Omron Sysmac Studio project OEEF_FS_lib_1_3_7 (Sysmac Studio 1.60.0.64010, LibraryProject)

# Controller new_Controller_0: NX1P2-1040DT1 version 1.21
Task PrimaryTask (priority 4, period or condition 2000): Programme0

TYPE nsAxisControl\eMoveMode : (Relative := 0, Absolute := 1); END_TYPE
TYPE nsAxisControl\eCurveType : (Poly5 := 0, Poly3 := 1, Straight := 2, NoCurve := 9999); END_TYPE
TYPE nsAxisControl\eTypeOfCmd : (CancelMC_Sync := -5, CancelCam := -3, CancelTrack := -2, NoCde := 9999, PolyMvt := 1, Track := 2, Cam := 3, WarmStart := 4, MC_Sync := 5); END_TYPE
TYPE nsAxisControl\stAxisControl : STRUCT
    MasterPosition : nsAxisControl\stMasterPosition;
    MasterAxis : _sAXIS_REF;
    Move : nsAxisControl\stMove;
    Track : nsAxisControl\stTrack;
    Cam : nsAxisControl\stCam;
    Flags : nsAxisControl\stFlags;
    Monitoring : nsAxisControl\stMonitoring;
    MC_MoveJog : nsAxisControl\stMC_MoveJog;
    MC_SetPosition : nsAxisControl\stMC_SetPosition;
    MC_Power : nsAxisControl\stMC_Power;
    MC_Home : nsAxisControl\stMC_Home;
END_STRUCT END_TYPE
TYPE nsAxisControl\stMC_Power : STRUCT
    Enable : BOOL;
    Status : BOOL;
    Busy : BOOL;
    Error : BOOL;
    ErrorID : WORD;
END_STRUCT END_TYPE
TYPE nsAxisControl\stMC_MoveJog : STRUCT
    PositiveEnable : BOOL;
    NegativeEnable : BOOL;
    Velocity : LREAL;
    Acceleration : LREAL;
    Deceleration : LREAL;
    Busy : BOOL;
    CommandAborted : BOOL;
    Error : BOOL;
    ErrorID : WORD;
END_STRUCT END_TYPE
TYPE nsAxisControl\stMC_SetPosition : STRUCT
    Execute : BOOL;
    Position : LREAL;
    ReferenceType : _eMC_REFERENCE_TYPE;
    Relative : BOOL;
    ExecutionMode : _eMC_EXECUTION_MODE;
    Done : BOOL;
    Busy : BOOL;
    CommandAborted : BOOL;
    Error : BOOL;
    ErrorID : WORD;
END_STRUCT END_TYPE
TYPE nsAxisControl\stMC_Home : STRUCT
    Execute : BOOL;
    Done : BOOL;
    Busy : BOOL;
    CommandAborted : BOOL;
    Error : BOOL;
    ErrorID : WORD;
END_STRUCT END_TYPE
TYPE nsAxisControl\stMasterPosition : STRUCT
    NotFrom_sAXIS_REF : BOOL;
    ExternalVariable : LREAL;
END_STRUCT END_TYPE
TYPE nsAxisControl\stMove : STRUCT
    Pos : LREAL;
    Dist : LREAL;
    Tim : LREAL;
    Accel : LREAL;
    Decel : LREAL;
    PolyType : nsAxisControl\eCurveType;
    Mode : nsAxisControl\eMoveMode;
    SetT_In : LREAL;
    SetT_Out : LREAL;
    T_InDone : BOOL;
    T_OutDone : BOOL;
    Exe : BOOL;
END_STRUCT END_TYPE
TYPE nsAxisControl\stTrack : STRUCT
    TrackPos : LREAL;
    Tim : LREAL;
    TimStop : LREAL;
    SetT_In : LREAL;
    T_InDone : BOOL;
    Exe : BOOL;
    Cancel : BOOL;
END_STRUCT END_TYPE
TYPE nsAxisControl\stCam : STRUCT
    Profile : ARRAY[0..10] OF nsAxisControl\stNodes;
    MasterOffset : LREAL;
    SlaveOffset : LREAL;
    ProfileToApply : INT;
    WarmStartSlavePos : LREAL;
    WarmStartSlavePosRequest : BOOL;
    Exe : BOOL;
    Cancel : BOOL;
END_STRUCT END_TYPE
TYPE nsAxisControl\stNodes : STRUCT
    Node : ARRAY[0..10] OF nsAxisControl\stNode;
END_STRUCT END_TYPE
TYPE nsAxisControl\stNode : STRUCT
    MasterAxisPos : LREAL;
    SlaveAxisPos : LREAL;
    CurveTypeBefore : nsAxisControl\eCurveType;
    StartingSlope : LREAL;
    EndingSlope : LREAL;
END_STRUCT END_TYPE
TYPE nsAxisControl\stFlags : STRUCT
    Done : BOOL;
    Synchronised : BOOL;
END_STRUCT END_TYPE
TYPE nsAxisControl\stMonitoring : STRUCT
    PositioningCmd : LREAL;
    CurrentProfile : INT;
    CurrentSegment : INT;
    TypeOfCmd : nsAxisControl\eTypeOfCmd;
END_STRUCT END_TYPE
TYPE nsAxisControl\eReferenceType : (mcCommand := 0, mcFeedback := 1); END_TYPE

PROGRAM Programme0

(* Section Section0: ladder, written here as Structured Text *)
END_PROGRAM

FUNCTION fPolyTimesNeeded : BOOL
(* - Time needed to achieve a movement depending of the curve type and the acceleration or the speed fixed. To do for instance a speed or an acceleration limit. *)
VAR_INPUT
    CurveType : nsAxisControl\eCurveType;
    Distance : LREAL;
    AccDefined : LREAL;
    SpeedDefined : LREAL;
END_VAR
VAR_OUTPUT
    TNeededToAcc : LREAL;
    TNeededToSpeed : LREAL;
END_VAR
(*
*******************************************
*		  Calcule le temps nécessaire			*
*	 pour effectuer un trajet avec une		*
*	accélération ou une vitesse définie		*
*******************************************
*)

CASE CurveType OF
	
	Poly5 :
	// AccDefined exprimée en unité/sec2
	TNeededToAcc:=SQRT(5.8*Distance/AccDefined);

	// SpeedDefined exprimée en unité/sec
	TNeededToSpeed:=1.9*Distance/SpeedDefined;
	
	Poly3 :
	// AccDefined exprimée en unité/sec2
	TNeededToAcc:=SQRT(6*Distance/AccDefined);

	// SpeedDefined exprimée en unité/sec
	TNeededToSpeed:=1.5*Distance/SpeedDefined;
	
END_CASE;
END_FUNCTION

FUNCTION fTicksQCalc : LINT
(* - Calculation of the quantity of ticks depending of the time of the movement *)
VAR
    TaskPeriod_msec : LINT;
END_VAR
VAR_INPUT
    TimeMvt : LREAL;
END_VAR
(*
*******************************************
*		  			Calcule le nombre				*
*	 					de cycles cpu					*
*******************************************
*)

// Suivant le temps de cycle de la tâche principale
TaskPeriod_msec:= TimeToNanoSec(GetMyTaskInterval())/1000000;

// Suivant le temps du mouvement en secondes
fTicksQCalc:=LREAL_TO_LINT(TimeMvt*1000)/TaskPeriod_msec;
END_FUNCTION

FUNCTION fPoly5 : LREAL
(* - Polynomial of the 5th order *)
VAR
    a : LREAL;
    b : LREAL;
    c : LREAL;
    d : LREAL;
    e : LREAL;
    f : LREAL;
    K : LREAL;
    xSq : LREAL;
END_VAR
VAR_INPUT
    v0 : LREAL;  (* Vitesse initiale *)
    v1 : LREAL;  (* Vitesse finale *)
    a0 : LREAL;
    a1 : LREAL;
    x : LREAL;
    Offset : LREAL;
    TargetDist : LREAL;
END_VAR
(*
*******************************************
*		  				Polynôme 5						*
*******************************************
*)

// Coéficients 
a:=6.0-3.0*(v0+v1)+((a1-a0)/2.0);
b:=-15.0+8.0*v0+7.0*v1+(3.0*a0/2.0)-a1;
c:=10.0-6.0*v0-4.0*v1-(3.0*a0/2.0)+(a1/2.0);
d:=a0/2.0;
e:=v0;
f:=Offset;
K:=TargetDist;

// Position=ax5+bx4+cx3+dx2+ex+f
fPoly5:=f+(K*(a*(x**5)+b*(x**4)+c*(x**3)+d*(x**2)+e*x));
END_FUNCTION

FUNCTION fPoly3 : LREAL
(* - Polynomial of the 3th order *)
VAR
    a : LREAL;
    b : LREAL;
    c : LREAL;
    d : LREAL;
    K : LREAL;
    xSq : LREAL;
END_VAR
VAR_INPUT
    v0 : LREAL;  (* Vitesse initiale *)
    v1 : LREAL;  (* Vitesse finale *)
    x : LREAL;
    Offset : LREAL;
    TargetDist : LREAL;
END_VAR
(*
*******************************************
*		  				Polynôme 3						*
*******************************************
*)

// Coéficients 
a:=-2.0+v0+v1;
b:=3.0-2.0*v0-v1;
c:=v0;
d:=Offset;
K:=TargetDist;

// Position=ax3+bx2+cx+d
fPoly3:=d+(K*(a*(x**3)+b*(x**2)+c*x));
END_FUNCTION

FUNCTION fStraight : LREAL
(* - Straight *)
VAR
    a : LREAL;
    b : LREAL;
END_VAR
VAR_INPUT
    x : LREAL;
    Offset : LREAL;
    TargetDist : LREAL;
END_VAR
(*
*******************************************
*		  					Droite							*
*******************************************
*)

// Coéficients 
a:=TargetDist;
b:=Offset;

// Position=ax+b
fStraight:=a*x+b;
END_FUNCTION

FUNCTION fAtan2 : LREAL
(* - Arc tangent on four quadrants *)
VAR
    PI : LREAL := 3.14159265358979;
END_VAR
VAR_INPUT
    x : LREAL;
    y : LREAL;
END_VAR
(*
*******************************************
*  Calcule l'arc tangente (angle en rad)	*
*  d'un point [x,y] dans les 4 quadrants	*
*******************************************
*)

IF x>0 THEN
	fAtan2:=ATAN(y/x);
ELSIF x<0 AND y>=0 THEN
	fAtan2:=ATAN(y/x)+PI;
ELSIF x<0 AND y<0 THEN
	fAtan2:=ATAN(y/x)-PI;
ELSIF x=0 AND y>0 THEN
	fAtan2:=PI/2;
ELSIF x=0 AND y<0 THEN
	fAtan2:=-PI/2;
ELSIF x=0 AND y=0 THEN
	fAtan2:=0.0; // Non défini
END_IF;
END_FUNCTION

FUNCTION_BLOCK AxisControl
(* - Cam on fly (multi-profiles) / - Warm start / - Polynomial moves / - Conveyor tracking / - Blending (T_In & T_Out) *)
VAR
    FBi_SyncMov : MC_SyncMoveAbsolute;
    FBi_SyncStop : MC_Stop;
    FBe_SetPosition : MC_SetPosition;
    FBe_Home : MC_Home;
    FBi_SyncMovVel : MC_SyncMoveVelocity;
    FBi_ReadAxisMasterParam : MC_ReadAxisParameter;
    FBi_ReadAxisSlaveParam : MC_ReadAxisParameter;
    FBe_Power : MC_Power;
    Edge1 : R_TRIG;
    Edge2 : R_TRIG;
    Edge3 : R_TRIG;
    Edge4 : R_TRIG;
    Edge5 : R_TRIG;
    Edge6 : R_TRIG;
    Edge10 : R_TRIG;
    TypeOfCmd : nsAxisControl\eTypeOfCmd;
    TargetDist : LREAL;
    UpExecMvt : BOOL;
    UpExecTrack : BOOL;
    UpExecCam : BOOL;
    UpCancelTrack : BOOL;
    Phase : INT;
    Tick : LINT;
    TicksQ : LINT;
    Offset : LREAL;
    x : LREAL;
    v0 : LREAL;  (* Vitesse initiale *)
    v1 : LREAL;  (* Vitesse finale *)
    DistStop : LREAL;
    UpCancelCam : BOOL;
    MasterDistDone : LREAL;
    a1 : LREAL;
    a0 : LREAL;
    FBe_MovJog : MC_MoveJog;
    MemPosAxis : LREAL;
    ReadAxisMasterPParam : _sAXIS_PARAM;
    ReadAxisSlavePParam : _sAXIS_PARAM;
    CamSettingError : BOOL;
    NodesNbMax : INT;
    Loop : INT;
    X0 : LREAL;
    X1 : LREAL;
    Y0 : LREAL;
    Y1 : LREAL;
    SegmentPolyType : nsAxisControl\eCurveType;
    MasterDist : LREAL;
    SegmentsNb : INT;
    NodesNb : INT;
    UpWarmStartPosReq : BOOL;
    WarmStartCalculation : BOOL;
    v1CamSetting : LREAL;
    v0CamSetting : LREAL;
    a0CamSetting : LREAL;
    a1CamSetting : LREAL;
    ScannedSeg : INT;
    SetPositionErr : BOOL;
    SetPositionErrID : WORD;
    CurrentProfile : INT := 0;
    ProfilesNb : INT;
    ProfilesNbMax : INT;
    UpCamBeginning : BOOL;
    CamSettingErrorType : STRING[50];
    Gen : LREAL;
    Conveyor_Pos : LREAL;
    TaskPeriod_msec_LREAL : LREAL;
    MasterPosition : LREAL;
    TickSetT_In : LINT;
    TickSetT_Out : LINT;
    memSegmentNb : INT;
    memPosition : LREAL;
    SlaveMinPos : LREAL;
    SlaveMaxPos : LREAL;
    SlaveCountMode : _eMC_COUNT_MODE;
    MasterModulo : LREAL;
    ReadAxisDelay : TON;
    SlaveModulo : LREAL;
    CurrentSegment : INT;
    CmdPos : LREAL;
    TargetSpeed : LREAL;
    FBi_dx : FB_dx_Codeur_V2;
    MasterMinPos : LREAL;
    MasterMaxPos : LREAL;
    dx : LREAL;
    MemSpeedAxis : LREAL;
    MemActPos : LREAL;
    TrackStopDelay : TON;
END_VAR
VAR_INPUT
    Reset : BOOL;
    ExternalError : BOOL;
END_VAR
VAR_OUTPUT
    Error : BOOL;
END_VAR
VAR_IN_OUT CONSTANT
    Axis : _sAXIS_REF;
END_VAR
VAR_IN_OUT
    IO : nsAxisControl\stAxisControl;
END_VAR
VAR_OUTPUT
    ErrorMsg : STRING[80];
END_VAR
(*
*******************************************
*					OEEF - F.SIMON					*
*******************************************
*)


(*
*******************************************
*	 		Bits fronts de statuts : RAZ			*
*******************************************
*)
IF IO.Flags.Done THEN
	IO.Flags.Done:=FALSE;
END_IF;

IF IO.Move.T_InDone THEN
	IO.Move.T_InDone:=FALSE;
END_IF;

IF IO.Move.T_OutDone THEN
	IO.Move.T_OutDone:=FALSE;
END_IF;

IF IO.Track.T_InDone THEN
	IO.Track.T_InDone:=FALSE;
END_IF;


(*
*******************************************
*						Axe maître						*
*******************************************
*)
// Type
IF IO.MasterPosition.NotFrom_sAXIS_REF THEN
	MasterPosition:=IO.MasterPosition.ExternalVariable;
ELSE
	MasterPosition:=IO.MasterAxis.Act.Pos;
END_IF;

// Offset
MasterModulo:=(ReadAxisSlavePParam.PosCount.ModuloMaxPosVal-ReadAxisSlavePParam.PosCount.ModuloMinPosVal);
IF IO.Cam.MasterOffset<0 THEN
	MasterPosition:=ModReal(MasterPosition-IO.Cam.MasterOffset,MasterModulo);
ELSE
	MasterPosition:=ModReal(MasterPosition+(MasterModulo-IO.Cam.MasterOffset),MasterModulo);
END_IF;


(*
*******************************************
*		Commande de tracking active		*
*******************************************
*)
// Etire le polynôme : recalcule la distance à parcourir depuis l'origine du tracking tant que l'on est pas synchronisé
IF TypeOfCmd=Track AND NOT IO.Flags.Synchronised THEN
	TargetDist:=IO.Track.TrackPos-MemPosAxis; 
END_IF;


(*
*******************************************
*			Commande 	de came					*
*			ou de warmstart active 				*
*******************************************
*)
IF TypeOfCmd=Cam OR TypeOfCmd=WarmStart THEN
	// Nombre de noeuds du profil
	NodesNb:=1;
	WHILE IO.Cam.Profile[CurrentProfile].Node[NodesNb].MasterAxisPos<>0
		DO
		NodesNb:=NodesNb+1;
	END_WHILE;

	// Nombre de segments
	SegmentsNb:=NodesNb-1;

	// Application du nouveau profil au passage du modulo du master en cas de changement à la volée
	IF MasterPosition<>memPosition THEN
		IF abs(memPosition-MasterPosition)>abs(MasterModulo)/2 THEN
			CurrentProfile:=IO.Cam.ProfileToApply;
		END_IF;
		memPosition:=MasterPosition;
	END_IF;	

	// Evolution du segment en cours
	FOR ScannedSeg:=0 TO SegmentsNb-1 DO
		IF MasterPosition>=IO.Cam.Profile[CurrentProfile].Node[ScannedSeg].MasterAxisPos AND MasterPosition<IO.Cam.Profile[CurrentProfile].Node[ScannedSeg+1].MasterAxisPos THEN
			CurrentSegment:=ScannedSeg;
		END_IF;
	END_FOR;

	// Paramètres du polynôme dans le segment en cours
	X0:=IO.Cam.Profile[CurrentProfile].Node[CurrentSegment].MasterAxisPos;											// Abscisse de début
	Y0:=IO.Cam.SlaveOffset+(IO.Cam.Profile[CurrentProfile].Node[CurrentSegment].SlaveAxisPos);			// Ordonnée de début
	X1:=IO.Cam.Profile[CurrentProfile].Node[CurrentSegment+1].MasterAxisPos;										// Abscisse de fin
	Y1:=IO.Cam.SlaveOffset+(IO.Cam.Profile[CurrentProfile].Node[CurrentSegment+1].SlaveAxisPos);		// Ordonnée de fin
	MasterDist:=X1-X0;																																	// Distance de la composante X
	TargetDist:=Y1-Y0;																																	// Distance de la composante Y
	Offset:=Y0;																																				// Offset de départ

	// Distance parcourue par le maître
	MasterDistDone:=MasterPosition-X0;
 
	SegmentPolyType:=IO.Cam.Profile[CurrentProfile].Node[CurrentSegment+1].CurveTypeBefore;		// Type de profil
	v0CamSetting:=IO.Cam.Profile[CurrentProfile].Node[CurrentSegment+1].StartingSlope;					// Pente de raccordement de la vitesse de début de segment
	v1CamSetting:=IO.Cam.Profile[CurrentProfile].Node[CurrentSegment+1].EndingSlope;					// Pente de raccordement de la vitesse de fin de segment
	//a0CamSetting:=?																																// Pente de raccordement de l'accélération de début de segment
	//a1CamSetting:=?																																// Pente de raccordement de l'accélération de fin de segment

	// Arrêt du calcul de la position de l'esclave pour le WarmStart
	IF WarmStartCalculation THEN
		WarmStartCalculation:=FALSE;
	END_IF;
END_IF;


(*
*******************************************
*						Générateur						*
*******************************************
*)
CASE Phase OF
	
	-1 : // ERREUR
	
		// Bits rémanents de statuts et de commandes : RAZ
		WarmStartCalculation:=FALSE;
		FBi_ReadAxisMasterParam.Execute:=FALSE;
		FBi_ReadAxisSlaveParam.Execute:=FALSE;
		FBi_SyncMov.Execute:=FALSE;
		FBi_SyncStop.Execute:=FALSE;
		FBi_SyncMovVel.Execute:=FALSE;
		IO.Flags.Synchronised:=FALSE;
	
		// Acquittement
		IF Error AND Reset THEN
			CamSettingError:=FALSE;
			Phase:=0;
		END_IF;
	
	0 : // COMMANDES

		IF NOT Error THEN
				Edge1(IO.Move.Exe,UpExecMvt);															// Commande de mouvement polynômial
				Edge2(IO.Track.Exe,UpExecTrack);														// Commande de tracking
				Edge3(IO.Track.Cancel,UpCancelTrack);												// Commande d'annulation de tracking
				Edge4(IO.Cam.Exe,UpExecCam);															// Commande de mise en came
				Edge5(IO.Cam.WarmStartSlavePosRequest,UpWarmStartPosReq);		// Commande de calcul de la position de l'esclave pour le WarmStart

				// Commande de mouvement polynômial
				IF UpExecMvt AND IO.Move.Tim>0 THEN
					TypeOfCmd:=PolyMvt;
					Gen:=Axis.Act.Pos;
					
					// Nombre de cycles cpu nécessaires pour le mouvement
					TicksQ:=fTicksQCalc(IO.Move.Tim);
					Tick:=0;
					
					// Calcul de la distance à effectuer
					IF IO.Move.Mode=Absolute THEN
						TargetDist:=IO.Move.Pos-Axis.Act.Pos;
					ELSIF IO.Move.Mode=Relative THEN
						TargetDist:=IO.Move.Dist;
					END_IF;
					
					Phase:=10;
				END_IF;
				
				// Commande de tracking
				IF UpExecTrack AND IO.Track.Tim>0 THEN
					TypeOfCmd:=Track;
					Gen:=Axis.Act.Pos;
					
					// Le début du tracking utilise une fonction polynômiale
					IO.Move.Tim:=IO.Track.Tim;
					// Nombre de cycles cpu nécessaires pour le mouvement
					TicksQ:=fTicksQCalc(IO.Track.Tim);
					Tick:=0;
					// Sauvegarde la position de l'axe
					MemPosAxis:=Axis.Act.Pos;
					// Calcul de la distance initiale à effectuer
					TargetDist:=IO.Track.TrackPos-MemPosAxis;
					Phase:=10;
				END_IF;
				
				// Commande d'annulation du tracking
				IF UpCancelTrack THEN
					TypeOfCmd:=CancelTrack;
					
					// Sauvegarde la vitesse de l'axe
					MemSpeedAxis:=Axis.Act.Vel;
					Phase:=30;
				END_IF;

				// Commande de came
				IF UpExecCam THEN
					TypeOfCmd:=Cam;
					Gen:=Axis.Act.Pos;
					
					ProfilesNbMax:=10;
					NodesNbMax:=10;
					CurrentProfile:=IO.Cam.ProfileToApply;
					CurrentSegment:=0;
					Phase:=5;
				END_IF;

				// Annulation de la commande de came : Traitée en Phase 20 pendant son exécution

				// Commande de calcul de la position de l'esclave pour le WarmStart
				IF UpWarmStartPosReq THEN
					TypeOfCmd:=WarmStart;
					ProfilesNbMax:=10;
					NodesNbMax:=10;
					CurrentProfile:=IO.Cam.ProfileToApply;
					CurrentSegment:=0;
					WarmStartCalculation:=TRUE;
					Phase:=5;
				END_IF;
		END_IF;


	5 : // INIT : lecture des paramètres des axes

		FBi_ReadAxisMasterParam.Execute:=TRUE;
		FBi_ReadAxisSlaveParam.Execute:=TRUE;
		
		IF FBi_ReadAxisMasterParam.Done AND FBi_ReadAxisSlaveParam.Done THEN
			ReadAxisDelay(In:=TRUE, PT:=T#10ms); // On s'assure que les paramètres sont propagés dans tout le FB
			IF ReadAxisDelay.Q THEN
				ReadAxisDelay(In:=FALSE);
				FBi_ReadAxisMasterParam.Execute:=FALSE;
				FBi_ReadAxisSlaveParam.Execute:=FALSE;
				Phase:=10;
			END_IF;
		ELSIF FBi_ReadAxisMasterParam.Error OR FBi_ReadAxisSlaveParam.Error THEN
			ReadAxisDelay(In:=FALSE);
			FBi_ReadAxisMasterParam.Execute:=FALSE;
			FBi_ReadAxisSlaveParam.Execute:=FALSE;
			Phase:=-1;
		END_IF;


	10 : // INIT : flags, offset
	
		// Exe
		FBi_SyncMov.Execute:=FALSE;
	
		// Distance nulle : on ne bouge pas
		IF abs(TargetDist)=0 THEN
			IO.Flags.Done:=TRUE;
			Phase:=0;
		END_IF;
		
		// Offsets de départ	
		IF TypeOfCmd<>Cam AND TypeOfCmd<>WarmStart THEN
			// Débute le mouvement à partir de la position actuelle
			Offset:=Axis.Act.Pos;
			Phase:=15;
		ELSIF TypeOfCmd=Cam THEN
			// Débute le mouvement à partir de Y0
			Offset:=Y0;
			Phase:=15;
		ELSIF TypeOfCmd=WarmStart THEN
			// Débute le mouvement à partir de Y0 et n'active pas la fonction de positionnement cyclique
			Offset:=Y0;
			Phase:=20;
		END_IF;
		
		
	15 : // INIT : activation de la fonction de positionnement cyclique
	
		FBi_SyncMov.Execute:=TRUE;
		
		IF FBi_SyncMov.Active THEN
			FBi_SyncMov.Execute:=FALSE;
			Phase:=20;
		ELSIF FBi_SyncMov.Error THEN
			FBi_SyncMov.Execute:=FALSE;
			Phase:=-1;
		END_IF;


	20 : // EXECUTION DU PROFIL

		// Flags
		IF TypeOfCmd=Cam THEN
			IO.Flags.Synchronised:=TRUE;		// En came
		END_IF;

		// Evolution de x
		//IF TypeOfCmd=PolyMvt OR TypeOfCmd=Track THEN
		IF TypeOfCmd=PolyMvt OR TypeOfCmd=Track THEN
			// En fonction du temps dans l'intervalle [0 ; 1] (hors came)
			x:=LIMIT(0.0,(1.0/LINT_TO_LREAL(TicksQ)*LINT_TO_LREAL(Tick)),1.0);
		ELSIF TypeOfCmd=Cam OR TypeOfCmd=WarmStart THEN
			// En fonction de la distance parcourue par le maître dans l'intervalle [0 ; 1] (En came)
			x:=LIMIT(0.0,((1.0/MasterDist)*MasterDistDone),1.0);
		END_IF;
		
		// Limites du domaine atteintes à 0,1 % et 99,9 % du parcours pour compenser les erreurs d'arrondis
		IF x<0.001 THEN
			x:=0;
		ELSIF x>0.999 THEN
			x:=1;
		END_IF;
		
		// Vitesses initiale et finale des polynômes 3 et 5
		IF TypeOfCmd=PolyMvt THEN
			 // Fixées à zéro pour un mouvement polynômial
			v0:=0.0;
			v1:=0.0;
		ELSIF TypeOfCmd=Track THEN
			// v1 en continuité avec celle du maître lors d'un tracking : elle est convertie dans l'intervalle [0;1] du polynôme EN COURS
			v0:=0.0;
			v1:=(1/(TargetDist/IO.Move.Tim))*IO.MasterAxis.Act.Vel;
		ELSIF TypeOfCmd=Cam OR TypeOfCmd=WarmStart THEN
			// Imposées par paramétrage de la came
			v0:=v0CamSetting;
			v1:=v1CamSetting;
		END_IF;
		
		// Accélérations initiale et finale du polynôme 5
		IF TypeOfCmd=PolyMvt THEN
			a0:=IO.Move.Accel;
			a1:=IO.Move.Decel;
		ELSIF TypeOfCmd=Cam OR TypeOfCmd=WarmStart THEN
			a0:=a0CamSetting;
			a1:=a1CamSetting;
		END_IF;
		
		// Polynôme 5
		IF TypeOfCmd=PolyMvt AND IO.Move.PolyType=Poly5
			OR
			(TypeOfCmd=Cam OR TypeOfCmd=WarmStart) AND SegmentPolyType=Poly5
			THEN
			Gen:=fPoly5(v0, v1, a0, a1, x, Offset, TargetDist);
		END_IF;

		// Polynôme 3
		IF TypeOfCmd=PolyMvt AND IO.Move.PolyType=Poly3 
			OR
			TypeOfCmd=Track 
			OR
			(TypeOfCmd=Cam OR TypeOfCmd=WarmStart) AND SegmentPolyType=Poly3
			THEN
			Gen:=fPoly3(v0, v1, x, Offset, TargetDist);
		END_IF;

		// Straight
		IF TypeOfCmd=PolyMvt AND IO.Move.PolyType=Straight 
			OR
			(TypeOfCmd=Cam OR TypeOfCmd=WarmStart) AND SegmentPolyType=Straight
			THEN
			Gen:=fStraight(x, Offset, TargetDist);
		END_IF;

		// Evolution du temps (hors came)
		IF TypeOfCmd=PolyMvt OR TypeOfCmd=Track THEN
			IF Tick<TicksQ THEN
				Inc(Tick);
	 		// Fin du polynome dans le cas d'une commande de type tracking
			ELSIF TypeOfCmd=Track THEN
				IO.Flags.Synchronised:=TRUE;
				IO.Flags.Done:=TRUE;
				Phase:=0;	
		 	// Fin du polynome dans le cas d'une commande de mouvement polynômial
			ELSIF TypeOfCmd=PolyMvt THEN
				Phase:=25;
			END_IF;
		END_IF;
		
		// Evolution du maître (en came)
		IF TypeOfCmd=Cam THEN			
			// Annulation de came
			Edge6(IO.Cam.Cancel,UpCancelCam);	
			IF UpCancelCam THEN
				IO.Flags.Synchronised:=FALSE;
				Phase:=25;
			END_IF;
		END_IF;
		
		// Calcul de la position de l'esclave pour le WarmStart
		IF TypeOfCmd=WarmStart THEN
			// Le calcul est terminé
			IO.Cam.WarmStartSlavePos:=Gen;
			IF NOT WarmStartCalculation THEN
				IO.Flags.Done:=TRUE;
				Phase:=0;
			END_IF;
		END_IF;
		
		
	25 : // DECONNEXION
	
		FBi_SyncStop.Execute:=TRUE;

		IF FBi_SyncStop.Done THEN
			FBi_SyncStop.Execute:=FALSE;			
			IO.Flags.Done:=TRUE;
			Phase:=0;
		ELSIF FBi_SyncStop.Error THEN
			FBi_SyncStop.Execute:=FALSE;
			Phase:=-1;			
		END_IF;
	
	
	30 : // DECELERATION LINEAIRE
	
		// Mode CSV à la dernière vitesse connue
		FBi_SyncMovVel.Velocity:=MemSpeedAxis;
		FBi_SyncMovVel.Execute:=TRUE;
		
		IF FBi_SyncMovVel.Busy THEN
			IO.Flags.Synchronised:=FALSE;
			FBi_SyncMovVel.Execute:=FALSE;
			// Taux de décélération
			FBi_SyncStop.Deceleration:=MemSpeedAxis/IO.Track.TimStop;
			Phase:=25;
		ELSIF FBi_SyncMovVel.Error THEN
			FBi_SyncMovVel.Execute:=FALSE;
			Phase:=-1;			
		END_IF;
	
END_CASE;


(*
*******************************************
*						Axe esclave						*
*******************************************
*)
SlaveMinPos:=ReadAxisSlavePParam.PosCount.ModuloMinPosVal;
SlaveMaxPos:=ReadAxisSlavePParam.PosCount.ModuloMaxPosVal;
SlaveModulo:=SlaveMaxPos-SlaveMinPos;
SlaveCountMode:=ReadAxisSlavePParam.PosCount.CountMode;
IF SlaveCountMode=_mcCountModeRotary THEN
	// Axe en modulo
	FBi_SyncMov.Direction:=_mcShortestWay;
	IF 	SlaveMinPos>=0 AND SlaveMaxPos>=0 THEN
		FBi_SyncMov.Position:=ABS(ModReal(Gen,SlaveModulo)); // Filtre la présence éventuelle de signe dans Gen
	ELSIF
		SlaveMinPos<0 AND SlaveMaxPos<0 THEN
		FBi_SyncMov.Position:=-1*(ABS(ModReal(Gen,SlaveModulo))); // Filtre l'absence éventuelle de signe dans Gen
		// Autre solution de filtrage : FBi_SyncMov.Position:=ModReal(Gen+SlaveModulo,SlaveModulo);
	ELSE
		FBi_SyncMov.Position:=ModReal(Gen,SlaveModulo);  // Pas de filtre : Gen négatif ou positif autorisé
	END_IF;	
ELSE
	// Axe en mode linéaire
	FBi_SyncMov.Direction:=_mcNoDirection;
	IF (TypeOfCmd=Track AND IO.Flags.Synchronised) OR TypeOfCmd=CancelTrack THEN
		// Polynôme de tracking terminé : synchronisation maître/esclave (following)
		FBi_SyncMov.Position:=IO.Track.TrackPos;
	ELSE
		FBi_SyncMov.Position:=Gen; // Pas de filtre : Gen négatif ou positif autorisé
	END_IF;
END_IF;


(*
*******************************************
*			T_InDone et T_OutDone				*
*******************************************
*)
// Délai atteint après le début d'un mouvement polynômial ou d'un tracking
TickSetT_In:=fTicksQCalc(IO.Move.SetT_In);
IF Tick=TickSetT_In THEN
	IF TypeOfCmd=PolyMvt THEN
		IO.Move.T_InDone:=TRUE;
	END_IF;
	IF TypeOfCmd=Track THEN
		IO.Track.T_InDone:=TRUE;
	END_IF;
END_IF;

// Délai atteint avant la fin d'un mouvement polynômial
TickSetT_Out:=fTicksQCalc(IO.Move.SetT_Out);
IF Tick=TickSetT_Out THEN
	IO.Move.T_OutDone:=TRUE;
END_IF;


(*
*******************************************
*	   Synthèse et messages d'erreurs		*
*******************************************
*)
// Synthèse des erreurs
IF FBi_SyncMov.Error OR FBi_SyncStop.Error OR FBi_ReadAxisMasterParam.Error OR FBi_ReadAxisSlaveParam.Error OR FBi_SyncMovVel.Error OR CamSettingError OR
	IO.MC_Power.Error OR IO.MC_MoveJog.Error OR IO.MC_SetPosition.Error OR IO.MasterAxis.MFaultLvl.Active OR IO.MasterAxis.Status.ErrorStop OR
	Axis.MFaultLvl.Active OR Axis.Status.ErrorStop OR ExternalError THEN
	Error:=TRUE;
	Phase:=-1;
ELSE
	Error:=FALSE;
END_IF;

// Erreur : l'axe maître n'est pas en mode rotationnel
IF (TypeOfCmd=Cam OR TypeOfCmd=WarmStart) THEN
	IF FBi_ReadAxisMasterParam.Done AND NOT (ReadAxisMasterPParam.PosCount.CountMode=_mcCountModeRotary) THEN
		CamSettingError:=TRUE;
		CamSettingErrorType:='Master axis is not in rotary count mode';
	END_IF;
END_IF;

// Erreur : le nombre de noeuds est supérieur au maximum autorisé
IF NodesNb>NodesNbMax THEN
	CamSettingError:=TRUE;
	CamSettingErrorType:='Too much nodes';
END_IF;

// Erreur : le nombre de profils est supérieur au maximum autorisé
IF ProfilesNb>ProfilesNbMax THEN
	CamSettingError:=TRUE;
	CamSettingErrorType:='Too much profiles';
END_IF;

// Erreur : une valeur maximale de modulo de l'axe maître a été franchie
IF IO.MasterAxis.Scale.CountMode=_mcCountModeRotary THEN
	FOR Loop:=0 TO NodesNb DO
		IF IO.Cam.Profile[CurrentProfile].Node[Loop].MasterAxisPos>IO.MasterAxis.Scale.MaxPos OR
			IO.Cam.Profile[CurrentProfile].Node[Loop].MasterAxisPos<IO.MasterAxis.Scale.MinPos THEN
			CamSettingError:=TRUE;
			CamSettingErrorType:='Master MaxPos or MinPos overflow';
		END_IF;
	END_FOR;
END_IF;

// Erreur : une valeur maximale de modulo de l'axe esclave a été franchie
IF Axis.Scale.CountMode=_mcCountModeRotary THEN
	FOR Loop:=0 TO NodesNb DO
		IF 	IO.Cam.Profile[CurrentProfile].Node[Loop].SlaveAxisPos+IO.Cam.SlaveOffset>Axis.Scale.MaxPos OR
			IO.Cam.Profile[CurrentProfile].Node[Loop].SlaveAxisPos+IO.Cam.SlaveOffset<Axis.Scale.MinPos THEN
			CamSettingError:=TRUE;
			CamSettingErrorType:='Slave MaxPos or MinPos overflow';
		END_IF;
	END_FOR;
END_IF;

// Erreur : une limite logicielle de l'axe maître a été franchie
IF ReadAxisMasterPParam.Limit.SwLimitMode<>_mcNonSwLmt THEN
	FOR Loop:=0 TO NodesNb DO
		IF 	IO.Cam.Profile[CurrentProfile].Node[Loop].MasterAxisPos>ReadAxisMasterPParam.Limit.PosiSwLimit OR
			IO.Cam.Profile[CurrentProfile].Node[Loop].MasterAxisPos<ReadAxisMasterPParam.Limit.NegaSwLimit THEN
			CamSettingError:=TRUE;
			CamSettingErrorType:='Master software limit overflow';
		END_IF;
	END_FOR;
END_IF;

// Erreur : une limite logicielle de l'axe esclave a été franchie
IF ReadAxisSlavePParam.Limit.SwLimitMode<>_mcNonSwLmt THEN
	FOR Loop:=0 TO NodesNb DO
		IF 	IO.Cam.Profile[CurrentProfile].Node[Loop].SlaveAxisPos>ReadAxisSlavePParam.Limit.PosiSwLimit OR
			IO.Cam.Profile[CurrentProfile].Node[Loop].SlaveAxisPos<ReadAxisSlavePParam.Limit.NegaSwLimit THEN
			CamSettingError:=TRUE;
			CamSettingErrorType:='Slave software limit overflow';
		END_IF;
	END_FOR;
END_IF;

// Messages d'erreur
IF FBi_SyncMov.Error THEN
	ErrorMsg:='Internal error : MC_SyncMoveAbsolute';
ELSIF
	FBi_SyncStop.Error THEN
	ErrorMsg:='Internal error : MC_Stop';
ELSIF
	FBi_ReadAxisMasterParam.Error THEN
	ErrorMsg:='Internal error : MC_ReadAxisParameter master';
ELSIF
	FBi_ReadAxisSlaveParam.Error THEN
	ErrorMsg:='Internal error : MC_ReadAxisParameter slave';
ELSIF
	FBi_SyncMovVel.Error THEN
	ErrorMsg:='Internal error : MC_SyncMoveVelocity';
ELSIF
	CamSettingError THEN
	ErrorMsg:=CONCAT('Internal error : Cam setting error ',CamSettingErrorType);
ELSIF
	IO.MC_Power.Error THEN
	ErrorMsg:='External error : MC_Power';
ELSIF
	IO.MC_MoveJog.Error THEN
	ErrorMsg:='External error : MC_MoveJog';
ELSIF
	IO.MC_SetPosition.Error THEN
	ErrorMsg:='External error : MC_SetPosition';
ELSIF
	IO.MasterAxis.MFaultLvl.Active OR IO.MasterAxis.Status.ErrorStop THEN
	ErrorMsg:='External error : Master minor or major error';
ELSIF
	Axis.MFaultLvl.Active OR Axis.Status.ErrorStop THEN
	ErrorMsg:='External error : Slave minor or major error';
ELSIF
	ExternalError THEN
	ErrorMsg:='External error : External error';
ELSE
	ClearString(ErrorMsg);
END_IF;
	

(*
*******************************************
*						Monitoring						*
*******************************************
*)
IO.Monitoring.PositioningCmd:=FBi_SyncMov.Position;
IO.Monitoring.TypeOfCmd:=TypeOfCmd;
IO.Monitoring.CurrentProfile:=CurrentProfile;		
IO.Monitoring.CurrentSegment:=CurrentSegment;


(*
*******************************************
*				Fonctions internes					*
*******************************************
*)
// Positionnement cyclique
FBi_SyncMov(
					Axis:=Axis, 
					BufferMode:=_mcAborting
					);

// Arrêt du positionnement cyclique
FBi_SyncStop(
					Axis:=Axis
					);

// Lecture des paramètres de l'axe maître
FBi_ReadAxisMasterParam(
					Axis:=IO.MasterAxis,
					AxisParameter:=ReadAxisMasterPParam
					);

// Lecture des paramètres de l'axe esclave
FBi_ReadAxisSlaveParam(
					Axis:=Axis,
					AxisParameter:=ReadAxisSlavePParam
					);

// MC_SyncMoveVelocity
FBi_SyncMovVel(
					Axis:=Axis
					);


(*
*******************************************
*				Fonctions externes					*
*******************************************
*)
// MC_Power
FBe_Power(
					Axis:=Axis, 
					Enable:=IO.MC_Power.Enable, 
					Status=>IO.MC_Power.Status, 
					Busy=>IO.MC_Power.Busy, 
					Error=>IO.MC_Power.Error, 
					ErrorID=>IO.MC_Power.ErrorID
					);

// MC_MoveJog
FBe_MovJog(
					Axis:= Axis,
					PositiveEnable:=IO.MC_MoveJog.PositiveEnable, 
					NegativeEnable:=IO.MC_MoveJog.NegativeEnable, 
					Velocity:=IO.MC_MoveJog.Velocity, 
					Acceleration:=IO.MC_MoveJog.Acceleration, 
					Deceleration:=IO.MC_MoveJog.Deceleration,
					Busy=>IO.MC_MoveJog.Busy, 
					CommandAborted=>IO.MC_MoveJog.CommandAborted, 
					Error=>IO.MC_MoveJog.Error, 
					ErrorID=>IO.MC_MoveJog.ErrorID
					);

// MC_SetPosition
FBe_SetPosition(
					Axis:=Axis,
					Execute:=IO.MC_SetPosition.Execute, 
					Position:=IO.MC_SetPosition.Position, 
					ReferenceType:=IO.MC_SetPosition.ReferenceType, 
					Relative:=IO.MC_SetPosition.Relative, 
					ExecutionMode:=IO.MC_SetPosition.ExecutionMode, 
					Done=>IO.MC_SetPosition.Done, 
					Busy=>IO.MC_SetPosition.Busy, 
					CommandAborted=>IO.MC_SetPosition.CommandAborted, 
					Error=>IO.MC_SetPosition.Error, 
					ErrorID=>IO.MC_SetPosition.ErrorID
					);

// MC_Home
FBe_Home(
					Axis:=Axis,
					Execute:=IO.MC_Home.Execute, 
					Done=>IO.MC_Home.Done, 
					Busy=>IO.MC_Home.Busy, 
					CommandAborted=>IO.MC_Home.CommandAborted, 
					Error=>IO.MC_Home.Error, 
					ErrorID=>IO.MC_Home.ErrorID
					);
	
END_FUNCTION_BLOCK

FUNCTION_BLOCK AverageFilter
(* - Makes an average filter of up to 100 samples *)
VAR
    Loop : INT;
    Samples : ARRAY[0..99] OF LREAL;
    Sum : LREAL;
END_VAR
VAR_INPUT
    Enable : BOOL;
END_VAR
VAR_OUTPUT
    Enabled : BOOL;
END_VAR
VAR_INPUT
    Measure : LREAL;
    QofSamples : INT;
END_VAR
VAR_OUTPUT
    Result : LREAL;
END_VAR
(*
*******************************************
*		   Filtre à moyenne glissante			*
*******************************************
*)

Loop:=1;
REPEAT
	// Pousse la pile pour libérer le premier rang
	Samples[QofSamples-Loop]:=Samples[QofSamples-(Loop+1)];
	Loop:=Loop+1;
UNTIL Loop>=QofSamples
END_REPEAT;
// Place le nouvel échantillon au premier rang
Samples[0]:=Measure;
Loop:=1;
Sum:=0.0;
REPEAT
	// Calcul la somme des échantillons
	Sum:=Sum+Samples[Loop-1];
	Loop:=Loop+1;
UNTIL Loop>QofSamples
END_REPEAT;
// Calcul la moyenne
Result:=Sum/QofSamples;
END_FUNCTION_BLOCK

FUNCTION_BLOCK FB_dx_Codeur_V2
(* - Provide the distance done per controller scan / - Manage the modulo's rollover in the two directions *)
VAR
    Mem_Position : LREAL;  (* Last position of the conveyor *)
    Max_Pos : LREAL;
END_VAR
VAR_INPUT
    Dummy : BOOL;
    Position : LREAL;  (* Position of the conveyor in mm *)
    Modulo_Max : LREAL;  (* Needed to handle overflow *)
    Modulo_Min : LREAL;  (* Needed to handle overflow *)
    Reverse : BOOL;  (* To reverse the signe of Delta_X *)
END_VAR
VAR_OUTPUT
    Delta_X : LREAL;
END_VAR
(*
***********************************
			FB_dx_Codeur_V2
***********************************
GP - Fevrier 2023
**********************************
Objet : 
- Le bloc transmet la vitesse / tour de scan du convoyeur
- Gère le rollOver du modulo dans les deux sens de marche
- Gère un modulo négatif et un modulo positif
***********************************

*)

Max_Pos := ABS(Modulo_Max - Modulo_Min);

// Calcul du dx 
Delta_X := Position - Mem_Position;
Mem_Position := Position;

// Cas du RollOver 
IF Delta_X <(-Max_Pos/2) THEN
	Delta_X := Delta_X + Max_Pos ;
END_IF;
IF Delta_X > (Max_Pos/2) THEN
	Delta_X := Delta_X - Max_Pos ;
END_IF;

IF Reverse THEN
	Delta_X := -1.0 * Delta_X;
END_IF;
END_FUNCTION_BLOCK

FUNCTION_BLOCK EncoderFilter
(* - Based on AverageFilter / - Makes a filtering of a modulo axis position *)
VAR
    Delta_X_Filtered : LREAL;
    Delta_X : LREAL;
    FB_dx_Encoder : FB_dx_Codeur_V2;
    FB_AverageFilter : AverageFilter;
    Position : LREAL;
END_VAR
VAR_INPUT
    Enable : BOOL;
    Axis : _sAXIS_REF;
    ReferenceType : nsAxisControl\eReferenceType;
    Modulo : LREAL;
    QofSamples : INT := 0;
END_VAR
VAR_OUTPUT
    Enabled : BOOL;
    Axis_Filtered : LREAL;
END_VAR
(* ladder, written here as Structured Text *)

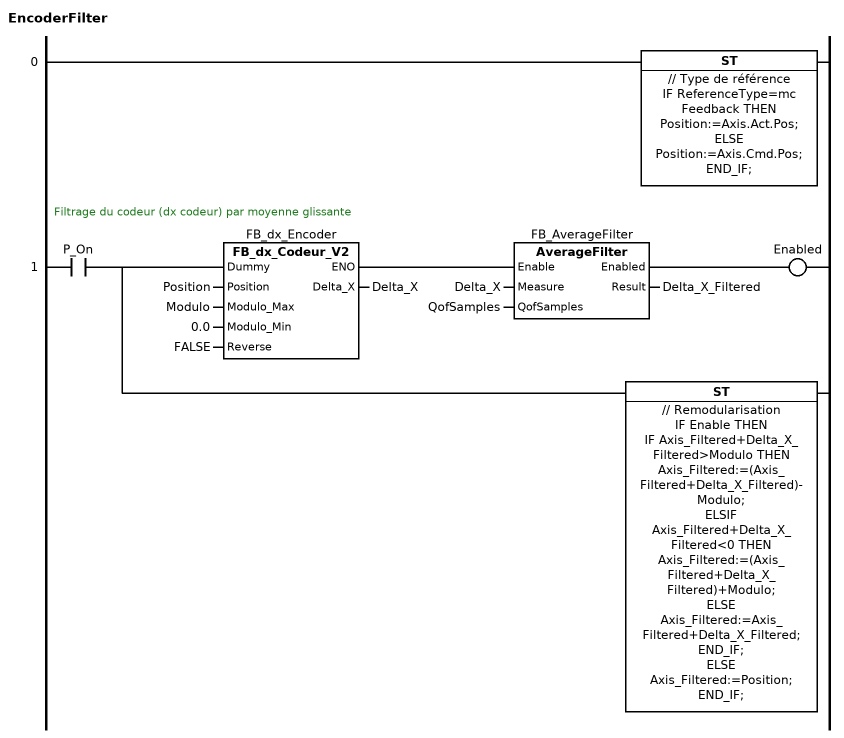
(* Rung 0 *)
// Type de référence
IF ReferenceType=mcFeedback THEN
	Position:=Axis.Act.Pos;
ELSE
	Position:=Axis.Cmd.Pos;
END_IF;
(* Rung 1: Filtrage du codeur (dx codeur) par moyenne glissante *)
FB_dx_Encoder(Dummy := P_On, Position := Position, Modulo_Max := Modulo, Modulo_Min := 0.0, Reverse := FALSE, Delta_X => Delta_X);
FB_AverageFilter(Enable := FB_dx_Encoder.ENO, Measure := Delta_X, QofSamples := QofSamples, Result => Delta_X_Filtered);
Enabled := FB_AverageFilter.Enabled;
IF P_On THEN
    // Remodularisation
    IF Enable THEN
    	IF Axis_Filtered+Delta_X_Filtered>Modulo THEN
    		Axis_Filtered:=(Axis_Filtered+Delta_X_Filtered)-Modulo;
    	ELSIF
    		Axis_Filtered+Delta_X_Filtered<0 THEN
    		Axis_Filtered:=(Axis_Filtered+Delta_X_Filtered)+Modulo;
    	ELSE
    		Axis_Filtered:=Axis_Filtered+Delta_X_Filtered;
    	END_IF;
    ELSE
    	Axis_Filtered:=Position;
    END_IF;
END_IF;
END_FUNCTION_BLOCK

FUNCTION_BLOCK FB_SysReset_V4
(* - Error reset of : PLC, Motion and Ethercat *)
VAR
    Index : UINT;
    State : INT;
    Init : BOOL;
    Nb_Axes : UINT;
    Nb_Groupes : UINT;
    Frm_Acquit : R_TRIG;
    Axis_Reset : BOOL;
    Group_Reset : BOOL;
    iFB_MC_Reset : MC_Reset;
    iFB_MC_ResetGroup : MC_GroupReset;
    iFB_ResetMC : ResetMCError;
    iFB_ResetEC : ResetECError;
    iFB_ResetPlc : ResetPLCError;
END_VAR
VAR_INPUT
    Reset : BOOL (* edge UpDirection *);
END_VAR
VAR_EXTERNAL CONSTANT
    _MC_AX : ARRAY[0..15] OF _sAXIS_REF;
    _MC_GRP : ARRAY[0..7] OF _sGROUP_REF;
END_VAR
(*
***********************************
				SysReset V4
***********************************
GP - Octobre 2013
**********************************
Objet : 
- Fonction permettant d'acquiter les défauts du systéme quelquesoit leur provenance
Le bloc intégre maintenant l'acquitement des axes et des groupes d'axes pour conserver l'exclusivité des blocs motion

Juillet 2015 : GP :  
	* Ajout du redémarrage du G7 sur une demande d'acquitement
	* Retrait des cartes CJB pour être compatible NX7
	
Decembre 2016 : GP :	Détecttion du nombre d'axes logiques et du nombre de groupe logique pour NX7 et NX1P
***********************************
*)

IF NOT Init THEN
	Nb_Axes := SizeOfAry(_MC_AX);
	Nb_Groupes := SizeOfAry(_MC_GRP);
	Init := TRUE;
END_IF;


Frm_Acquit(CLK:=Reset);
IF Frm_Acquit.Q THEN 
	State:=0;
END_IF;

CASE State OF 
	
0 : 	(* Attente demande d'acquitement *)

	iFB_ResetEC (Execute := FALSE);
	iFB_ResetMC (Execute := FALSE);
	iFB_ResetPlc (Execute := FALSE);
	
	Axis_Reset := FALSE;
	Group_Reset := FALSE;
	
	IF Reset THEN
		State := 10;
	END_IF;
		
10: (* Parcours de tous les axes pour les acquitter *)	
	 
	 Index := 0;
	 State := 20;
	 
20: (* Test si l'axe est utilisé *)
 
	 IF  _MC_AX[Index].Cfg.AxEnable = _mcUsedAxis THEN
		 Axis_Reset := TRUE;
		 State := 30;
	 ELSE
		 State := 40;
	 END_IF;
	 
30: (* Attente que l'axe soit réseter *)
	
	IF iFB_MC_Reset.Done THEN
		Axis_Reset := FALSE;
		State := 40;
	END_IF;
	
40 : (* Incrémentation de l'index *)

	Inc(Index);
	
	IF Index < Nb_Axes THEN
		State := 20;
	ELSE
		State := 50;
	END_IF;
	
50: (* Parcours de tous les groupes pour les acquitter *)	
	 
	 Index := 0;
	 State := 60;
	 
60: (* Test si l'axe est utilisé *)
	 
	 IF _MC_GRP[Index].Cfg.GrpEnable = _mcUsedGroup THEN
		Group_Reset := TRUE;
		 State := 70;
	 ELSE
	 	State := 80;
	 END_IF;
	 
70: (* Attente que le groupe soit réseter *)
	
	IF iFB_MC_ResetGroup.Done THEN
		Group_Reset := FALSE;
		State := 80;
	END_IF;
	
80 : (* Incrémentation de l'index *)

	Inc(Index);
	
	IF Index < Nb_Groupes THEN
		State := 60;
	ELSE
		State := 90;
	END_IF;
	
90 : (* Acquitement du Motion Controler *)

	iFB_ResetMC (Execute := TRUE);

	IF iFB_ResetMC.Done THEN
		iFB_ResetMC (Execute := FALSE);
		State := 100;
	END_IF;

100 : (* Acquitement des alarmes utilisateurs *)
	
	IF GetAlarm() THEN
		ResetAlarm(0);
	END_IF;
	
	State := 110;
	
110 : (* Acquitement du maitre Ethercat *)
	
	iFB_ResetEC (Execute := TRUE);

	IF iFB_ResetEC.Done THEN
		iFB_ResetEC (Execute := FALSE);
		State := 120;
	END_IF;	
	
120 : (* Reset de la CPU *)

	iFB_ResetPlc (Execute := TRUE);
	
	IF iFB_ResetPlc.Done THEN
		iFB_ResetPlc (Execute := FALSE);
		State := 0;
	END_IF;
	
END_CASE;

(* Gestion des FBs *)
 iFB_MC_Reset(Axis:= _MC_AX[Index], Execute:= Axis_Reset);
 iFB_MC_ResetGroup(AxesGroup:= _MC_GRP[Index], Execute:= Group_Reset);
END_FUNCTION_BLOCK